{attribute 'qualified_only'}
{attribute 'strict'}
TYPE EAbortState :
(
	none := 0,
	requested := 1,
	aborting := 2,
	aborted := 3
);
END_TYPE

(* stored: Version 1.1.0.1, ProductVersion 3.1.4024.12
   DUT EAbortState: Id {fa29e679-eb35-4388-b046-483355300658} *)
